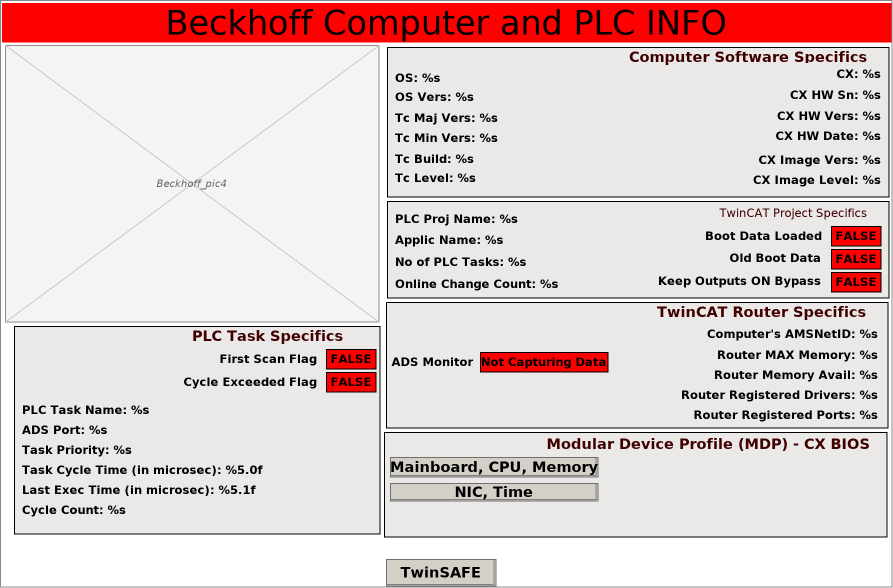
VISUALIZATION TwinCAT_INFO  // 893x588
    RoundedRectangle (384,432 503x105)
    Button (386,559 110x27), "TwinSAFE"
        OnMouseClick: change screen: TwinSAFE
    RoundedRectangle (2,3 889x39), "Beckhoff Computer and PLC INFO"
    RoundedRectangle (387,47 502x150)
    Label (614,44 256x26), "Computer Software Specifics"
    Rectangle (392,67 256x22), "OS: %s", text variable: g_stHMI_DevIdent.strImageOsName
    RoundedRectangle (387,201 502x97)
    Label (695,200 175x26), "TwinCAT Project Specifics"
    RoundedRectangle (386,302 502x126)
    Label (613,299 256x26), "TwinCAT Router Specifics"
    RoundedRectangle (14,326 366x208)
    Label (188,323 158x26), "PLC Task Specifics"
    Rectangle (392,86 208x22), "OS Vers: %s", text variable: g_stHMI_DevIdent.strImageOsVersion
    Rectangle (392,107 119x22), "Tc Maj Vers: %s", text variable: g_stHMI_DevIdent.strTwinCATVersion
    Rectangle (392,127 111x22), "Tc Min Vers: %s", text variable: g_stHMI_DevIdent.strTwinCATRevision
    Rectangle (392,148 111x22), "Tc Build: %s", text variable: g_stHMI_DevIdent.strTwinCATBuild
    Rectangle (392,167 111x22), "Tc Level: %s", text variable: g_stHMI_DevIdent.strTwinCATLevel
    Rectangle (738,63 146x22), "CX: %s", text variable: g_stHMI_DevIdent.strHardwareModel
    Rectangle (726,84 158x22), "CX HW Sn: %s", text variable: g_stHMI_DevIdent.strHardwareSerialNo
    Rectangle (733,105 151x22), "CX HW Vers: %s", text variable: g_stHMI_DevIdent.strHardwareVersion
    Rectangle (737,125 147x22), "CX HW Date: %s", text variable: g_stHMI_DevIdent.strHardwareDate
    Rectangle (725,149 159x22), "CX Image Vers: %s", text variable: g_stHMI_DevIdent.strImageVersion
    Rectangle (625,169 259x22), "CX Image Level: %s", text variable: g_stHMI_DevIdent.strImageLevel
    Rectangle (392,208 283x22), "PLC Proj Name: %s", text variable: g_stHMI_AppInfo.ProjectName
    Rectangle (392,229 359x22), "Applic Name: %s", text variable: g_stHMI_AppInfo.AppName
    Rectangle (392,251 155x22), "No of PLC Tasks: %s", text variable: g_stHMI_AppInfo.TaskCnt
    Rectangle (392,273 191x22), "Online Change Count: %s", text variable: g_stHMI_AppInfo.OnlineChangeCnt
    Group (831,226 50x20)
        Rectangle (0,0 50x20), "TRUE", invisible if: NOT g_stHMI_AppInfo.BootDataLoaded
        Rectangle (0,0 50x20), "FALSE", invisible if: g_stHMI_AppInfo.BootDataLoaded
    Label (705,224 120x24), "Boot Data Loaded"
    Group (831,249 50x20)
        Rectangle (0,0 50x20), "TRUE", invisible if: NOT g_stHMI_AppInfo.OldBootData
        Rectangle (0,0 50x20), "FALSE", invisible if: g_stHMI_AppInfo.OldBootData
    Label (726,246 98x24), "Old Boot Data"
    Group (831,272 50x20)
        Rectangle (0,0 49x19), "TRUE", invisible if: NOT g_stHMI_AppInfo.KeepOutputsOnBP
        Rectangle (0,0 50x20), "FALSE", invisible if: g_stHMI_AppInfo.KeepOutputsOnBP
    Label (645,269 179x24), "Keep Outputs ON Bypass"
    Label (389,350 87x24), "ADS Monitor"
    Group (480,352 128x20)
        Rectangle (0,0 128x20), "Capturing Data", invisible if: NOT g_stHMI_RouterStatusInfo.amsDebugLog
        Rectangle (0,0 128x20), "Not Capturing Data", invisible if: g_stHMI_RouterStatusInfo.amsDebugLog
    Rectangle (560,323 321x22), "Computer's AMSNetID: %s", text variable: g_stHMI_DevIdent.strAmsNetId
    Rectangle (673,344 208x22), "Router MAX Memory: %s", text variable: g_stHMI_RouterStatusInfo.maxMem
    Rectangle (673,364 208x22), "Router Memory Avail: %s", text variable: g_stHMI_RouterStatusInfo.maxMemAvail
    Rectangle (673,384 208x22), "Router Registered Drivers: %s", text variable: g_stHMI_RouterStatusInfo.regDrivers
    Rectangle (673,404 208x22), "Router Registered Ports: %s", text variable: g_stHMI_RouterStatusInfo.regPorts
    Group (326,349 50x20)
        Rectangle (0,0 50x20), "TRUE", invisible if: NOT g_stHMI_PlcTaskSystemInfo.FirstCycle
        Rectangle (0,0 50x20), "FALSE", invisible if: g_stHMI_PlcTaskSystemInfo.FirstCycle
    Label (200,347 120x24), "First Scan Flag"
    Group (326,372 50x20)
        Rectangle (0,0 50x20), "TRUE", invisible if: NOT g_stHMI_PlcTaskSystemInfo.CycleTimeExceeded
        Rectangle (0,0 50x20), "FALSE", invisible if: g_stHMI_PlcTaskSystemInfo.CycleTimeExceeded
    Label (178,370 142x24), "Cycle Exceeded Flag"
    Rectangle (19,399 357x22), "PLC Task Name: %s", text variable: g_stHMI_PlcTaskSystemInfo.TaskName
    Rectangle (19,419 299x22), "ADS Port: %s", text variable: g_stHMI_PlcTaskSystemInfo.AdsPort
    Rectangle (19,439 214x22), "Task Priority: %s", text variable: g_stHMI_PlcTaskSystemInfo.Priority
    Rectangle (19,459 298x22), "Task Cycle Time (in microsec): %5.0f", text variable: g_lrHMI_PlcTaskSystemInfo_CycleTime
    Rectangle (19,479 298x22), "Last Exec Time (in microsec): %5.1f", text variable: g_lrHMI_PlcTaskSystemInfo_LastExecTime
    Rectangle (19,499 214x22), "Cycle Count: %s", text variable: g_stHMI_PlcTaskSystemInfo.CycleCount
    Button (390,483 208x18), "NIC, Time"
        OnMouseClick: change screen: MDP_NicTime
    Button (390,457 208x20), "Mainboard, CPU, Memory"
        OnMouseClick: change screen: MDP_MainboardCPUMemory
    Label (516,431 357x26), "Modular Device Profile (MDP) - CX BIOS"
    Image (5,45 374x277), image: Beckhoff_pic4
END_VISUALIZATION

(* stored: Version 1.1.0.1, ProductVersion 3.1.0.18
   Visu TwinCAT_INFO: Id {319d32cd-6358-4f17-a08d-5447f8085241} *)
